FUNCTION_BLOCK FB_Utilities_Dispatcher
VAR_INPUT
	i_cooling_pump_req : ST_Util_Service_Req;
	i_deadair_pump_req : ST_Util_Service_Req;
END_VAR
VAR_OUTPUT
	o_cooling_pump_assigned : BOOL;
	o_deadair_pump_assigned : BOOL;
END_VAR

VAR
	cooling_pump_dispatch : FB_Service_Dispatcher();
	deadair_pump_dispatch : FB_Service_Dispatcher();
END_VAR




cooling_pump_dispatch( i_service_req := i_cooling_pump_req, o_service_assigned_sts => o_cooling_pump_assigned);
deadair_pump_dispatch( i_service_req := i_deadair_pump_req, o_service_assigned_sts => o_deadair_pump_assigned);

END_FUNCTION_BLOCK

(* stored: Version 1.1.0.1, ProductVersion 3.1.4024.12
   POU FB_Utilities_Dispatcher: Id {d0755d92-1ccf-48ac-9a0e-e752bed1f7d0}, SpecialFunc None *)
